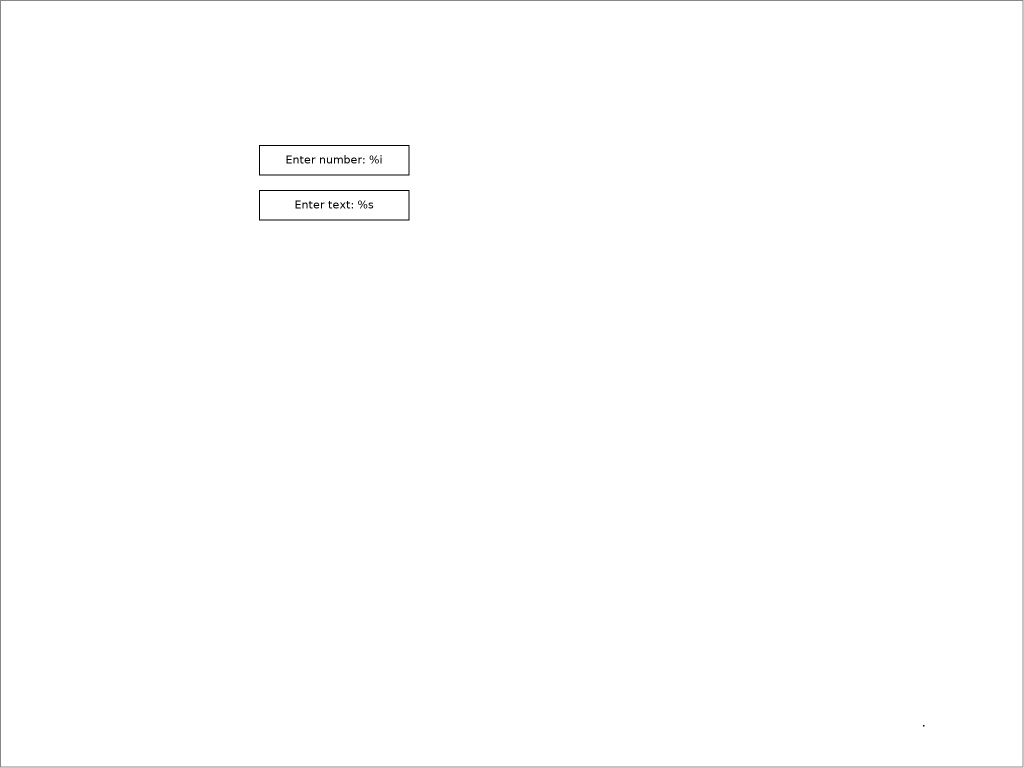
VISUALIZATION Visualization  // 1024x768
    Rectangle (259,145 150x30), "Enter number: %i", text variable: MAIN.iTest
        OnMouseDown: write the text variable via Default
    Rectangle (259,190 150x30), "Enter text: %s", text variable: MAIN.sTest
        OnMouseDown: write the text variable via Default
    Rectangle (923,725 1x1)
END_VISUALIZATION

(* stored: Version 1.1.0.1, ProductVersion 3.1.4024.3
   Visu Visualization: Id {7aefb3c9-5bfe-47ea-ba72-49647123698f} *)
